// TIA Portal V20 export
DATA_BLOCK "db_1"   // DB1
{ S7_Optimized_Access := 'TRUE' }
// stored: MemoryReserve 100
   VAR
      var_1 : Bool;
      var_2 { ExternalAccessible := 'False'; ExternalVisible := 'False'; ExternalWritable := 'False'} : Int;
      var_3 : Real;
   END_VAR
   VAR RETAIN
      var_4 : Array[0..9] of Bool;
   END_VAR
   VAR
      var_5 { ExternalWritable := 'False'} : Struct
         var_5_1 : Bool;
         var_5_2 : Int;
         var_5_3 : Real;
      END_STRUCT;
      var_6 { S7_SetPoint := 'True'} : Bool;
      var_7 { ExternalVisible := 'False'} : Real;
      var_8 : IEC_COUNTER;
      var_9 : IEC_TIMER;
   END_VAR
BEGIN
END_DATA_BLOCK
